FUNCTION_BLOCK Wait
VAR_OUTPUT
    Klaar 	: BOOL 	:= FALSE;
END_VAR

VAR
    Tmr 	: TON;
    Running : BOOL 	:= FALSE;
	flase	: BOOL;
	done	: BOOL;
END_VAR

// Timer automatisch starten zodra FB wordt opgeroepen en wacht 5s tot klaar = true

Tmr(IN := TRUE, PT := T#5S);
IF Done = TRUE THEN
	klaar := FALSE;
	tmr(IN := FALSE);
	Done := FALSE;
END_IF
IF Tmr.Q THEN
	done := TRUE;
	klaar := TRUE;
END_IF

END_FUNCTION_BLOCK

(* stored: Version 1.1.0.1, ProductVersion 3.1.4024.15
   POU Wait: Id {c6ca6f8d-7df5-4b31-aba1-c53ed20e65c8}, SpecialFunc None *)
